(* IEC 61131-3 sources: stc/stdlib/vendor/allen_bradley, 3 files *)

(* ---- instructions.st ---- *)
(* Allen Bradley Logix 5000 -- Common instruction stubs *)
(* These map AB instruction mnemonics to IEC FUNCTION declarations. *)
(* AB uses these as instructions; stc stubs them as functions for type-checking. *)

(* Arithmetic instructions *)
FUNCTION ADD : DINT
VAR_INPUT
    SourceA     : DINT;
    SourceB     : DINT;
END_VAR
END_FUNCTION

FUNCTION SUB : DINT
VAR_INPUT
    SourceA     : DINT;
    SourceB     : DINT;
END_VAR
END_FUNCTION

FUNCTION MUL : DINT
VAR_INPUT
    SourceA     : DINT;
    SourceB     : DINT;
END_VAR
END_FUNCTION

FUNCTION DIV : DINT
VAR_INPUT
    SourceA     : DINT;
    SourceB     : DINT;
END_VAR
END_FUNCTION

(* Data move instruction *)
FUNCTION MOV : DINT
VAR_INPUT
    Source      : DINT;
END_VAR
END_FUNCTION

(* Comparison instructions -- return BOOL for condition evaluation *)
FUNCTION CMP : BOOL
VAR_INPUT
    Expression  : STRING(80);
END_VAR
END_FUNCTION

FUNCTION EQU : BOOL
VAR_INPUT
    SourceA     : DINT;
    SourceB     : DINT;
END_VAR
END_FUNCTION

FUNCTION NEQ : BOOL
VAR_INPUT
    SourceA     : DINT;
    SourceB     : DINT;
END_VAR
END_FUNCTION

FUNCTION GRT : BOOL
VAR_INPUT
    SourceA     : DINT;
    SourceB     : DINT;
END_VAR
END_FUNCTION

FUNCTION LES : BOOL
VAR_INPUT
    SourceA     : DINT;
    SourceB     : DINT;
END_VAR
END_FUNCTION

FUNCTION GEQ : BOOL
VAR_INPUT
    SourceA     : DINT;
    SourceB     : DINT;
END_VAR
END_FUNCTION

FUNCTION LEQ : BOOL
VAR_INPUT
    SourceA     : DINT;
    SourceB     : DINT;
END_VAR
END_FUNCTION

(* ---- profile.st ---- *)
(* Allen Bradley Logix 5000 -- AB-compatible type stubs *)
(* AB restrictions: no OOP, no POINTER TO, no REFERENCE TO, tag-based I/O *)
(* These stubs use standard IEC 61131-3 FUNCTION_BLOCK syntax. *)
(* The stc checker uses the AB vendor profile to restrict language features. *)

(* AB timer accumulator type used by TONR, TOFR, RTO *)
TYPE TIMER :
STRUCT
    PRE         : DINT;     (* Preset value in milliseconds *)
    ACC         : DINT;     (* Accumulated value in milliseconds *)
    EN          : BOOL;     (* Timer enable bit *)
    TT          : BOOL;     (* Timer timing bit *)
    DN          : BOOL;     (* Timer done bit *)
END_STRUCT
END_TYPE

(* AB counter type *)
TYPE COUNTER :
STRUCT
    PRE         : DINT;     (* Preset value *)
    ACC         : DINT;     (* Accumulated value *)
    CU          : BOOL;     (* Count up enable *)
    CD          : BOOL;     (* Count down enable *)
    DN          : BOOL;     (* Done bit *)
    OV          : BOOL;     (* Overflow bit *)
    UN          : BOOL;     (* Underflow bit *)
END_STRUCT
END_TYPE

(* AB CONTROL structure for block transfer and other instructions *)
TYPE CONTROL :
STRUCT
    LEN         : DINT;     (* Length *)
    POS         : DINT;     (* Position *)
    EN          : BOOL;     (* Enable *)
    EU          : BOOL;     (* Enable unload *)
    DN          : BOOL;     (* Done *)
    EM          : BOOL;     (* Empty *)
    ER          : BOOL;     (* Error *)
    FD          : BOOL;     (* Found *)
    IN_         : BOOL;     (* Inhibit *)
    UL          : BOOL;     (* Unload *)
END_STRUCT
END_TYPE

(* AB MSG instruction for peer-to-peer communication *)
FUNCTION_BLOCK MSG
VAR_INPUT
    Execute     : BOOL;
    MsgType     : DINT;
    TargetAddr  : STRING(80);
    LocalTag    : STRING(80);
    RemoteTag   : STRING(80);
END_VAR
VAR_OUTPUT
    EN          : BOOL;
    DN          : BOOL;
    ER          : BOOL;
    ErrorCode   : DINT;
END_VAR
END_FUNCTION_BLOCK

(* ---- timers.st ---- *)
(* Allen Bradley Logix 5000 -- Timer instruction stubs *)
(* AB uses different timer names and behavior from IEC standard *)

(* TONR -- Timer On Delay Retentive *)
(* Unlike IEC TON, TONR retains accumulated time when disabled *)
FUNCTION_BLOCK TONR
VAR_INPUT
    TimerEnable : BOOL;
    PRE         : DINT;     (* Preset value in milliseconds *)
END_VAR
VAR_OUTPUT
    ACC         : DINT;     (* Accumulated value in milliseconds *)
    EN          : BOOL;     (* Timer enable bit *)
    TT          : BOOL;     (* Timer timing bit *)
    DN          : BOOL;     (* Timer done bit *)
END_VAR
END_FUNCTION_BLOCK

(* TOFR -- Timer Off Delay Retentive *)
FUNCTION_BLOCK TOFR
VAR_INPUT
    TimerEnable : BOOL;
    PRE         : DINT;     (* Preset value in milliseconds *)
END_VAR
VAR_OUTPUT
    ACC         : DINT;     (* Accumulated value *)
    EN          : BOOL;
    TT          : BOOL;
    DN          : BOOL;
END_VAR
END_FUNCTION_BLOCK

(* RTO -- Retentive Timer On *)
(* Accumulates time while enabled, retains value when disabled *)
(* Must be explicitly reset with RES instruction *)
FUNCTION_BLOCK RTO
VAR_INPUT
    TimerEnable : BOOL;
    PRE         : DINT;     (* Preset value in milliseconds *)
END_VAR
VAR_OUTPUT
    ACC         : DINT;     (* Accumulated value *)
    EN          : BOOL;
    TT          : BOOL;
    DN          : BOOL;
END_VAR
END_FUNCTION_BLOCK
